(*
  Managing software requirements
*)
FUNCTION_BLOCK FB_SRS
VAR
  nSrsCt   : UDINT := 0;
  sSrsList : ARRAY[1..100] OF ST_SRS :=  // (software) requirements list
  [
    (bImplemented:=TRUE, skey:='first srs', sDescription:='first detail', sLink:='https://polytype.atlassian.net/browse/STWE-71')    
  ];
  
  bInit : BOOL;
END_VAR

(*
  Show a list of implemented SRS software/machine requirements. 
  Best linked to JIRA-Tiuckets, OPL or Steinmann Smartsheet entries.
*)

IF NOT bInit THEN
  bInit := TRUE;
END_IF

END_FUNCTION_BLOCK

(* stored: Version 1.1.0.1, ProductVersion 3.1.4024.11
   POU FB_SRS: Id {f196b89b-aa46-4ad1-8386-42e56422aa0c}, SpecialFunc None *)
